LIN {X 0,Y 216.642,Z 888.332,A -85,B 0,C 180,E1 18460.085,E2 18460.085} C_VEL
LIN {X 0,Y 215.367,Z 897.562,A -85,B 0,C 180,E1 18472.801,E2 18472.801} C_VEL
LIN {X 0,Y 221.756,Z 891.791,A -85,B 0,C 180,E1 18485.568,E2 18485.568} C_VEL
LIN {X 0,Y 234.367,Z 872.004,A -85,B 0,C 180,E1 18496.083,E2 18496.083} C_VEL
LIN {X 0,Y 246.425,Z 844.143,A -85,B 0,C 180,E1 18503.35,E2 18503.35} C_VEL
LIN {X 0,Y 242.463,Z 813.223,A -85,B 0,C 180,E1 18511.998,E2 18511.998} C_VEL
LIN {X 0,Y 229.534,Z 783.44,A -85,B 0,C 180,E1 18522.815,E2 18522.815} C_VEL
LIN {X 0,Y 219.501,Z 768.602,A -85,B 0,C 180,E1 18532.547,E2 18532.547} C_VEL
LIN {X 0,Y 216.132,Z 762.311,A -85,B 0,C 180,E1 18538.989,E2 18538.989} C_VEL
LIN {X 0,Y 216.801,Z 764.753,A -85,B 0,C 180,E1 18552.68,E2 18552.68} C_VEL
LIN {X 0,Y 226.089,Z 777.855,A -85,B 0,C 180,E1 18563.686,E2 18563.686} C_VEL
LIN {X 0,Y 243.459,Z 806.862,A -85,B 0,C 180,E1 18574.796,E2 18574.796} C_VEL
LIN {X 0,Y 255.396,Z 841.876,A -85,B 0,C 180,E1 18582.72,E2 18582.72} C_VEL
LIN {X 0,Y 253.54,Z 855.895,A -85,B 0,C 180,E1 18584.51,E2 18584.51} C_VEL
LIN {X 0,Y 237.346,Z 898.415,A -85,B 0,C 180,E1 18590.848,E2 18590.848} C_VEL
LIN {X 0,Y 221.071,Z 933.004,A -85,B 0,C 180,E1 18601.282,E2 18601.282} C_VEL
LIN {X 0,Y 213.369,Z 954.07,A -85,B 0,C 180,E1 18614.546,E2 18614.546} C_VEL
LIN {X 0,Y 214.082,Z 960.88,A -85,B 0,C 180,E1 18627.97,E2 18627.97} C_VEL
LIN {X 0,Y 213.585,Z 955.524,A -85,B 0,C 180,E1 18638.754,E2 18638.754} C_VEL
LIN {X 0,Y 215.65,Z 935.355,A -85,B 0,C 180,E1 18651.683,E2 18651.683} C_VEL
LIN {X 0,Y 225.142,Z 901.268,A -85,B 0,C 180,E1 18662.599,E2 18662.599} C_VEL
LIN {X 0,Y 236.885,Z 857.02,A -85,B 0,C 180,E1 18669.903,E2 18669.903} C_VEL
LIN {X 0,Y 239.376,Z 834.505,A -85,B 0,C 180,E1 18672.297,E2 18672.297} C_VEL
LIN {X 0,Y 223.033,Z 785.451,A -85,B 0,C 180,E1 18678.284,E2 18678.284} C_VEL
LIN {X 0,Y 208.065,Z 754.81,A -85,B 0,C 180,E1 18683.186,E2 18683.186} C_VEL
LIN {X 0,Y 208.631,Z 754.81,A -85,B 0,C 180,E1 18696.424,E2 18696.424} C_VEL
LIN {X 0,Y 209.987,Z 754.81,A -85,B 0,C 180,E1 18709.596,E2 18709.596} C_VEL
LIN {X 0,Y 211.028,Z 754.81,A -85,B 0,C 180,E1 18722.066,E2 18722.066} C_VEL
LIN {X 0,Y 209.557,Z 754.81,A -85,B 0,C 180,E1 18734.688,E2 18734.688} C_VEL
LIN {X 0,Y 208.363,Z 754.81,A -85,B 0,C 180,E1 18748.262,E2 18748.262} C_VEL
LIN {X 0,Y 207.688,Z 754.81,A -85,B 0,C 180,E1 18755.24,E2 18755.24} C_VEL
LIN {X 0,Y 199.559,Z 754.81,A -85,B 0,C 180,E1 18765.026,E2 18765.026} C_VEL
LIN {X 0,Y 200.085,Z 754.81,A -85,B 0,C 180,E1 18780.729,E2 18780.729} C_VEL
LIN {X 0,Y 200.76,Z 756.849,A -85,B 0,C 180,E1 18786.458,E2 18786.458} C_VEL
LIN {X 0,Y 219.95,Z 797.875,A -85,B 0,C 180,E1 18793.889,E2 18793.889} C_VEL
LIN {X 0,Y 225.128,Z 832.107,A -85,B 0,C 180,E1 18800.297,E2 18800.297} C_VEL
LIN {X 0,Y 216.024,Z 866.137,A -85,B 0,C 180,E1 18808.489,E2 18808.489} C_VEL
LIN {X 0,Y 208.947,Z 888.832,A -85,B 0,C 180,E1 18819.404,E2 18819.404} C_VEL
LIN {X 0,Y 207.037,Z 897.624,A -85,B 0,C 180,E1 18829.258,E2 18829.258} C_VEL
LIN {X 0,Y 211.47,Z 896.323,A -85,B 0,C 180,E1 18842.561,E2 18842.561} C_VEL
LIN {X 0,Y 222.672,Z 881.638,A -85,B 0,C 180,E1 18853.742,E2 18853.742} C_VEL
LIN {X 0,Y 238.779,Z 852.504,A -85,B 0,C 180,E1 18862.854,E2 18862.854} C_VEL
LIN {X 0,Y 239.096,Z 827.128,A -85,B 0,C 180,E1 18870.117,E2 18870.117} C_VEL
LIN {X 0,Y 230.039,Z 797.834,A -85,B 0,C 180,E1 18880.234,E2 18880.234} C_VEL
LIN {X 0,Y 218.96,Z 777.151,A -85,B 0,C 180,E1 18891.777,E2 18891.777} C_VEL
LIN {X 0,Y 214.743,Z 770.093,A -85,B 0,C 180,E1 18899.995,E2 18899.995} C_VEL
LIN {X 0,Y 215.607,Z 772.884,A -85,B 0,C 180,E1 18912.422,E2 18912.422} C_VEL
LIN {X 0,Y 224.315,Z 785.804,A -85,B 0,C 180,E1 18923.242,E2 18923.242} C_VEL
LIN {X 0,Y 239.528,Z 813.168,A -85,B 0,C 180,E1 18934.071,E2 18934.071} C_VEL
LIN {X 0,Y 249.646,Z 846.608,A -85,B 0,C 180,E1 18942.026,E2 18942.026} C_VEL
LIN {X 0,Y 234.399,Z 890.534,A -85,B 0,C 180,E1 18948.112,E2 18948.112} C_VEL
LIN {X 0,Y 217.163,Z 925.879,A -85,B 0,C 180,E1 18957.631,E2 18957.631} C_VEL
LIN {X 0,Y 206.591,Z 949.509,A -85,B 0,C 180,E1 18970.699,E2 18970.699} C_VEL
LIN {X 0,Y 205.64,Z 959.398,A -85,B 0,C 180,E1 18984.976,E2 18984.976} C_VEL
LIN {X 0,Y 205.897,Z 956.427,A -85,B 0,C 180,E1 18996.349,E2 18996.349} C_VEL
LIN {X 0,Y 206.874,Z 939.032,A -85,B 0,C 180,E1 19009.834,E2 19009.834} C_VEL
LIN {X 0,Y 215.884,Z 906.703,A -85,B 0,C 180,E1 19021.819,E2 19021.819} C_VEL
LIN {X 0,Y 227.99,Z 864.284,A -85,B 0,C 180,E1 19029.883,E2 19029.883} C_VEL
LIN {X 0,Y 232.17,Z 835.979,A -85,B 0,C 180,E1 19033.141,E2 19033.141} C_VEL
LIN {X 0,Y 216.478,Z 787.844,A -85,B 0,C 180,E1 19039.468,E2 19039.468} C_VEL
LIN {X 0,Y 200.012,Z 754.81,A -85,B 0,C 180,E1 19045.323,E2 19045.323} C_VEL
LIN {X 0,Y 201.013,Z 754.81,A -85,B 0,C 180,E1 19060.687,E2 19060.687} C_VEL
LIN {X 0,Y 202.403,Z 754.81,A -85,B 0,C 180,E1 19073.548,E2 19073.548} C_VEL
LIN {X 0,Y 202.353,Z 754.81,A -85,B 0,C 180,E1 19086.465,E2 19086.465} C_VEL
LIN {X 0,Y 200.993,Z 754.81,A -85,B 0,C 180,E1 19099.868,E2 19099.868} C_VEL
LIN {X 0,Y 199.695,Z 754.81,A -85,B 0,C 180,E1 19115.187,E2 19115.187} C_VEL
LIN {X 0,Y 199.559,Z 754.81,A -85,B 0,C 180,E1 19125.026,E2 19125.026} C_VEL
LIN {X 0,Y 191.609,Z 754.81,A -85,B 0,C 180,E1 19135.197,E2 19135.197} C_VEL
LIN {X 0,Y 192.38,Z 756.459,A -85,B 0,C 180,E1 19144.182,E2 19144.182} C_VEL
LIN {X 0,Y 211.999,Z 796.756,A -85,B 0,C 180,E1 19152.184,E2 19152.184} C_VEL
LIN {X 0,Y 217.973,Z 830.392,A -85,B 0,C 180,E1 19158.773,E2 19158.773} C_VEL
LIN {X 0,Y 209.876,Z 862.822,A -85,B 0,C 180,E1 19166.371,E2 19166.371} C_VEL
LIN {X 0,Y 201.767,Z 887.669,A -85,B 0,C 180,E1 19177.517,E2 19177.517} C_VEL
LIN {X 0,Y 199.152,Z 899.09,A -85,B 0,C 180,E1 19190.053,E2 19190.053} C_VEL
LIN {X 0,Y 204.345,Z 897.187,A -85,B 0,C 180,E1 19203.846,E2 19203.846} C_VEL
LIN {X 0,Y 217.901,Z 879.987,A -85,B 0,C 180,E1 19216.181,E2 19216.181} C_VEL
LIN {X 0,Y 233.671,Z 850.1,A -85,B 0,C 180,E1 19225.187,E2 19225.187} C_VEL
LIN {X 0,Y 231.584,Z 820.81,A -85,B 0,C 180,E1 19234.506,E2 19234.506} C_VEL
LIN {X 0,Y 221.936,Z 794.694,A -85,B 0,C 180,E1 19245.77,E2 19245.77} C_VEL
LIN {X 0,Y 214.394,Z 778.368,A -85,B 0,C 180,E1 19257.967,E2 19257.967} C_VEL
LIN {X 0,Y 214.31,Z 780.597,A -85,B 0,C 180,E1 19271.92,E2 19271.92} C_VEL
LIN {X 0,Y 222.449,Z 793.997,A -85,B 0,C 180,E1 19282.967,E2 19282.967} C_VEL
LIN {X 0,Y 235.748,Z 820.234,A -85,B 0,C 180,E1 19293.604,E2 19293.604} C_VEL
LIN {X 0,Y 243.852,Z 851.713,A -85,B 0,C 180,E1 19301.417,E2 19301.417} C_VEL
LIN {X 0,Y 226.095,Z 894.862,A -85,B 0,C 180,E1 19307.709,E2 19307.709} C_VEL
LIN {X 0,Y 207.49,Z 930.206,A -85,B 0,C 180,E1 19318.594,E2 19318.594} C_VEL
LIN {X 0,Y 198.097,Z 950.734,A -85,B 0,C 180,E1 19332.015,E2 19332.015} C_VEL
LIN {X 0,Y 197.56,Z 957.948,A -85,B 0,C 180,E1 19343.385,E2 19343.385} C_VEL
LIN {X 0,Y 198.021,Z 956.031,A -85,B 0,C 180,E1 19355.118,E2 19355.118} C_VEL
LIN {X 0,Y 198.683,Z 939.873,A -85,B 0,C 180,E1 19369.188,E2 19369.188} C_VEL
LIN {X 0,Y 207.133,Z 909.933,A -85,B 0,C 180,E1 19381.469,E2 19381.469} C_VEL
LIN {X 0,Y 219.913,Z 867.584,A -85,B 0,C 180,E1 19390.314,E2 19390.314} C_VEL
LIN {X 0,Y 225.138,Z 838.311,A -85,B 0,C 180,E1 19393.92,E2 19393.92} C_VEL
LIN {X 0,Y 210.626,Z 791.691,A -85,B 0,C 180,E1 19400.501,E2 19400.501} C_VEL
LIN {X 0,Y 191.887,Z 754.81,A -85,B 0,C 180,E1 19406.991,E2 19406.991} C_VEL
LIN {X 0,Y 192.724,Z 754.81,A -85,B 0,C 180,E1 19419.253,E2 19419.253} C_VEL
LIN {X 0,Y 194.322,Z 754.81,A -85,B 0,C 180,E1 19433.279,E2 19433.279} C_VEL
LIN {X 0,Y 194.279,Z 754.81,A -85,B 0,C 180,E1 19446.734,E2 19446.734} C_VEL
LIN {X 0,Y 192.8,Z 754.81,A -85,B 0,C 180,E1 19460.75,E2 19460.75} C_VEL
LIN {X 0,Y 191.639,Z 754.81,A -85,B 0,C 180,E1 19476.442,E2 19476.442} C_VEL
LIN {X 0,Y 191.645,Z 754.81,A -85,B 0,C 180,E1 19493.564,E2 19493.564} C_VEL
LIN {X 0,Y 191.609,Z 754.81,A -85,B 0,C 180,E1 19495.197,E2 19495.197} C_VEL
LIN {X 0,Y 183.731,Z 754.81,A -85,B 0,C 180,E1 19499.208,E2 19499.208} C_VEL
LIN {X 0,Y 184.236,Z 756.635,A -85,B 0,C 180,E1 19501.717,E2 19501.717} C_VEL
LIN {X 0,Y 203.8,Z 794.802,A -85,B 0,C 180,E1 19510.168,E2 19510.168} C_VEL
LIN {X 0,Y 210.927,Z 830.344,A -85,B 0,C 180,E1 19517.504,E2 19517.504} C_VEL
LIN {X 0,Y 204.215,Z 859.007,A -85,B 0,C 180,E1 19524.134,E2 19524.134} C_VEL
LIN {X 0,Y 194.675,Z 886.406,A -85,B 0,C 180,E1 19535.591,E2 19535.591} C_VEL
LIN {X 0,Y 191.171,Z 899.454,A -85,B 0,C 180,E1 19548.437,E2 19548.437} C_VEL
LIN {X 0,Y 195.686,Z 899.486,A -85,B 0,C 180,E1 19562.877,E2 19562.877} C_VEL
LIN {X 0,Y 208.51,Z 885.123,A -85,B 0,C 180,E1 19575.477,E2 19575.477} C_VEL
LIN {X 0,Y 225.786,Z 857.601,A -85,B 0,C 180,E1 19584.905,E2 19584.905} C_VEL
LIN {X 0,Y 227.56,Z 833.221,A -85,B 0,C 180,E1 19592.776,E2 19592.776} C_VEL
LIN {X 0,Y 221.295,Z 807.811,A -85,B 0,C 180,E1 19603.05,E2 19603.05} C_VEL
LIN {X 0,Y 213.936,Z 790.965,A -85,B 0,C 180,E1 19614.525,E2 19614.525} C_VEL
LIN {X 0,Y 212.043,Z 785.811,A -85,B 0,C 180,E1 19621.02,E2 19621.02} C_VEL
LIN {X 0,Y 212.903,Z 788.641,A -85,B 0,C 180,E1 19631.751,E2 19631.751} C_VEL
LIN {X 0,Y 220.234,Z 801.886,A -85,B 0,C 180,E1 19642.689,E2 19642.689} C_VEL
LIN {X 0,Y 231.995,Z 827.726,A -85,B 0,C 180,E1 19653.366,E2 19653.366} C_VEL
LIN {X 0,Y 237.051,Z 855.918,A -85,B 0,C 180,E1 19660.426,E2 19660.426} C_VEL
LIN {X 0,Y 217.838,Z 898.908,A -85,B 0,C 180,E1 19667.307,E2 19667.307} C_VEL
LIN {X 0,Y 199.27,Z 931.565,A -85,B 0,C 180,E1 19678.429,E2 19678.429} C_VEL
LIN {X 0,Y 189.619,Z 951.846,A -85,B 0,C 180,E1 19693.734,E2 19693.734} C_VEL
LIN {X 0,Y 190.23,Z 957.232,A -85,B 0,C 180,E1 19707.715,E2 19707.715} C_VEL
LIN {X 0,Y 189.591,Z 950.728,A -85,B 0,C 180,E1 19720.377,E2 19720.377} C_VEL
LIN {X 0,Y 193.25,Z 928.656,A -85,B 0,C 180,E1 19734.969,E2 19734.969} C_VEL
LIN {X 0,Y 204.698,Z 893.624,A -85,B 0,C 180,E1 19746.379,E2 19746.379} C_VEL
LIN {X 0,Y 217.917,Z 847.797,A -85,B 0,C 180,E1 19753.779,E2 19753.779} C_VEL
LIN {X 0,Y 209.733,Z 808.336,A -85,B 0,C 180,E1 19759.633,E2 19759.633} C_VEL
LIN {X 0,Y 186.372,Z 760.571,A -85,B 0,C 180,E1 19768.233,E2 19768.233} C_VEL
LIN {X 0,Y 183.924,Z 754.81,A -85,B 0,C 180,E1 19770.042,E2 19770.042} C_VEL
LIN {X 0,Y 185.05,Z 754.81,A -85,B 0,C 180,E1 19783.326,E2 19783.326} C_VEL
LIN {X 0,Y 186.802,Z 754.81,A -85,B 0,C 180,E1 19797.678,E2 19797.678} C_VEL
LIN {X 0,Y 185.727,Z 754.81,A -85,B 0,C 180,E1 19811.793,E2 19811.793} C_VEL
LIN {X 0,Y 184.071,Z 754.81,A -85,B 0,C 180,E1 19826.971,E2 19826.971} C_VEL
LIN {X 0,Y 183.347,Z 754.81,A -85,B 0,C 180,E1 19844.72,E2 19844.72} C_VEL
LIN {X 0,Y 183.731,Z 754.81,A -85,B 0,C 180,E1 19859.208,E2 19859.208} C_VEL
LIN {X 0,Y 186.245,Z 763.492,A -85,B 0,C 180,E1 19862.685,E2 19862.685} C_VEL
LIN {X 0,Y 191.204,Z 782.709,A -85,B 0,C 180,E1 19865.652,E2 19865.652} C_VEL
LIN {X 0,Y 202.789,Z 819.29,A -85,B 0,C 180,E1 19873.694,E2 19873.694} C_VEL
LIN {X 0,Y 201.736,Z 846.339,A -85,B 0,C 180,E1 19879.748,E2 19879.748} C_VEL
LIN {X 0,Y 190.445,Z 878.405,A -85,B 0,C 180,E1 19890.153,E2 19890.153} C_VEL
LIN {X 0,Y 183.865,Z 896.903,A -85,B 0,C 180,E1 19903.118,E2 19903.118} C_VEL
LIN {X 0,Y 184.797,Z 902.481,A -85,B 0,C 180,E1 19916.849,E2 19916.849} C_VEL
LIN {X 0,Y 195.151,Z 894.31,A -85,B 0,C 180,E1 19931.374,E2 19931.374} C_VEL
LIN {X 0,Y 212.21,Z 872.098,A -85,B 0,C 180,E1 19942.65,E2 19942.65} C_VEL
LIN {X 0,Y 221.528,Z 853.18,A -85,B 0,C 180,E1 19948.193,E2 19948.193} C_VEL
LIN {X 0,Y 220.459,Z 825.911,A -85,B 0,C 180,E1 19958.323,E2 19958.323} C_VEL
LIN {X 0,Y 213.555,Z 802.898,A -85,B 0,C 180,E1 19970.794,E2 19970.794} C_VEL
LIN {X 0,Y 210.375,Z 793.636,A -85,B 0,C 180,E1 19980.929,E2 19980.929} C_VEL
LIN {X 0,Y 211.106,Z 796.544,A -85,B 0,C 180,E1 19991.517,E2 19991.517} C_VEL
LIN {X 0,Y 217.693,Z 809.685,A -85,B 0,C 180,E1 20002.449,E2 20002.449} C_VEL
LIN {X 0,Y 227.555,Z 834.107,A -85,B 0,C 180,E1 20012.806,E2 20012.806} C_VEL
LIN {X 0,Y 231.22,Z 857.687,A -85,B 0,C 180,E1 20019.123,E2 20019.123} C_VEL
LIN {X 0,Y 211.548,Z 899.02,A -85,B 0,C 180,E1 20025.984,E2 20025.984} C_VEL
LIN {X 0,Y 191.672,Z 931.777,A -85,B 0,C 180,E1 20037.696,E2 20037.696} C_VEL
LIN {X 0,Y 181.601,Z 951.475,A -85,B 0,C 180,E1 20053.923,E2 20053.923} C_VEL
LIN {X 0,Y 182.292,Z 956.015,A -85,B 0,C 180,E1 20067.616,E2 20067.616} C_VEL
LIN {X 0,Y 181.721,Z 950.328,A -85,B 0,C 180,E1 20079.616,E2 20079.616} C_VEL
LIN {X 0,Y 184.679,Z 930.394,A -85,B 0,C 180,E1 20094.23,E2 20094.23} C_VEL
LIN {X 0,Y 196.232,Z 896.463,A -85,B 0,C 180,E1 20106.48,E2 20106.48} C_VEL
LIN {X 0,Y 209.934,Z 852.254,A -85,B 0,C 180,E1 20114.357,E2 20114.357} C_VEL
LIN {X 0,Y 209.002,Z 831.793,A -85,B 0,C 180,E1 20117.414,E2 20117.414} C_VEL
LIN {X 0,Y 193.105,Z 786.695,A -85,B 0,C 180,E1 20124.963,E2 20124.963} C_VEL
LIN {X 0,Y 176.04,Z 754.81,A -85,B 0,C 180,E1 20132.545,E2 20132.545} C_VEL
LIN {X 0,Y 177.688,Z 754.81,A -85,B 0,C 180,E1 20149.175,E2 20149.175} C_VEL
LIN {X 0,Y 178.858,Z 754.81,A -85,B 0,C 180,E1 20162.438,E2 20162.438} C_VEL
LIN {X 0,Y 177.009,Z 754.81,A -85,B 0,C 180,E1 20177.468,E2 20177.468} C_VEL
LIN {X 0,Y 175.399,Z 754.81,A -85,B 0,C 180,E1 20194.717,E2 20194.717} C_VEL
LIN {X 0,Y 175.178,Z 754.81,A -85,B 0,C 180,E1 20209.477,E2 20209.477} C_VEL
LIN {X 0,Y 175.877,Z 756.396,A -85,B 0,C 180,E1 20218.796,E2 20218.796} C_VEL
LIN {X 0,Y 191.204,Z 782.709,A -85,B 0,C 180,E1 20225.652,E2 20225.652} C_VEL
LIN {X 0,Y 194.539,Z 813.73,A -85,B 0,C 180,E1 20230.805,E2 20230.805} C_VEL
LIN {X 0,Y 196.081,Z 842.903,A -85,B 0,C 180,E1 20237.716,E2 20237.716} C_VEL
LIN {X 0,Y 184.277,Z 875.529,A -85,B 0,C 180,E1 20247.639,E2 20247.639} C_VEL
LIN {X 0,Y 176.592,Z 896.01,A -85,B 0,C 180,E1 20260.798,E2 20260.798} C_VEL
LIN {X 0,Y 176.358,Z 903.64,A -85,B 0,C 180,E1 20275.361,E2 20275.361} C_VEL
LIN {X 0,Y 186.16,Z 897.498,A -85,B 0,C 180,E1 20290.699,E2 20290.699} C_VEL
LIN {X 0,Y 204.093,Z 876.474,A -85,B 0,C 180,E1 20303.025,E2 20303.025} C_VEL
LIN {X 0,Y 215.35,Z 856.378,A -85,B 0,C 180,E1 20309.262,E2 20309.262} C_VEL
LIN {X 0,Y 215.666,Z 832.062,A -85,B 0,C 180,E1 20318.855,E2 20318.855} C_VEL
LIN {X 0,Y 210.513,Z 809.89,A -85,B 0,C 180,E1 20331.432,E2 20331.432} C_VEL
LIN {X 0,Y 208.183,Z 801.185,A -85,B 0,C 180,E1 20342.083,E2 20342.083} C_VEL
LIN {X 0,Y 208.98,Z 804.42,A -85,B 0,C 180,E1 20351.385,E2 20351.385} C_VEL
LIN {X 0,Y 214.51,Z 816.583,A -85,B 0,C 180,E1 20361.797,E2 20361.797} C_VEL
LIN {X 0,Y 222.765,Z 839.779,A -85,B 0,C 180,E1 20372.04,E2 20372.04} C_VEL
LIN {X 0,Y 224.498,Z 861.643,A -85,B 0,C 180,E1 20378.011,E2 20378.011} C_VEL
LIN {X 0,Y 203.15,Z 902.913,A -85,B 0,C 180,E1 20385.548,E2 20385.548} C_VEL
LIN {X 0,Y 183.452,Z 932.959,A -85,B 0,C 180,E1 20397.474,E2 20397.474} C_VEL
LIN {X 0,Y 173.684,Z 950.664,A -85,B 0,C 180,E1 20413.637,E2 20413.637} C_VEL
LIN {X 0,Y 174.339,Z 954.776,A -85,B 0,C 180,E1 20427.507,E2 20427.507} C_VEL
LIN {X 0,Y 173.756,Z 948.862,A -85,B 0,C 180,E1 20440.062,E2 20440.062} C_VEL
LIN {X 0,Y 177.417,Z 927.956,A -85,B 0,C 180,E1 20455.624,E2 20455.624} C_VEL
LIN {X 0,Y 189.677,Z 893.977,A -85,B 0,C 180,E1 20467.959,E2 20467.959} C_VEL
LIN {X 0,Y 203.64,Z 850.097,A -85,B 0,C 180,E1 20475.748,E2 20475.748} C_VEL
LIN {X 0,Y 196.001,Z 811.221,A -85,B 0,C 180,E1 20482.437,E2 20482.437} C_VEL
LIN {X 0,Y 174.661,Z 766.987,A -85,B 0,C 180,E1 20491.859,E2 20491.859} C_VEL
LIN {X 0,Y 168.178,Z 754.81,A -85,B 0,C 180,E1 20496.05,E2 20496.05} C_VEL
LIN {X 0,Y 170.064,Z 754.81,A -85,B 0,C 180,E1 20512.314,E2 20512.314} C_VEL
LIN {X 0,Y 170.796,Z 754.81,A -85,B 0,C 180,E1 20522.553,E2 20522.553} C_VEL
LIN {X 0,Y 168.649,Z 754.81,A -85,B 0,C 180,E1 20539.115,E2 20539.115} C_VEL
LIN {X 0,Y 167.173,Z 754.81,A -85,B 0,C 180,E1 20556.169,E2 20556.169} C_VEL
LIN {X 0,Y 167.158,Z 754.81,A -85,B 0,C 180,E1 20573.833,E2 20573.833} C_VEL
LIN {X 0,Y 168.298,Z 758.387,A -85,B 0,C 180,E1 20575.922,E2 20575.922} C_VEL
LIN {X 0,Y 187.651,Z 792.072,A -85,B 0,C 180,E1 20585.695,E2 20585.695} C_VEL
LIN {X 0,Y 194.539,Z 813.73,A -85,B 0,C 180,E1 20590.805,E2 20590.805} C_VEL
LIN {X 0,Y 191.602,Z 836.321,A -85,B 0,C 180,E1 20595.002,E2 20595.002} C_VEL
LIN {X 0,Y 189.261,Z 843.612,A -85,B 0,C 180,E1 20596.494,E2 20596.494} C_VEL
LIN {X 0,Y 176.72,Z 876.776,A -85,B 0,C 180,E1 20606.922,E2 20606.922} C_VEL
LIN {X 0,Y 168.388,Z 898.052,A -85,B 0,C 180,E1 20621.546,E2 20621.546} C_VEL
LIN {X 0,Y 168.057,Z 904.57,A -85,B 0,C 180,E1 20633.974,E2 20633.974} C_VEL
LIN {X 0,Y 177.177,Z 900.405,A -85,B 0,C 180,E1 20649.969,E2 20649.969} C_VEL
LIN {X 0,Y 195.65,Z 881.029,A -85,B 0,C 180,E1 20663.258,E2 20663.258} C_VEL
LIN {X 0,Y 209.024,Z 860.383,A -85,B 0,C 180,E1 20670.037,E2 20670.037} C_VEL
LIN {X 0,Y 210.464,Z 835.648,A -85,B 0,C 180,E1 20680.514,E2 20680.514} C_VEL
LIN {X 0,Y 206.875,Z 814.753,A -85,B 0,C 180,E1 20693.677,E2 20693.677} C_VEL
LIN {X 0,Y 205.811,Z 808.827,A -85,B 0,C 180,E1 20702.107,E2 20702.107} C_VEL
LIN {X 0,Y 206.426,Z 811.438,A -85,B 0,C 180,E1 20710.585,E2 20710.585} C_VEL
LIN {X 0,Y 212.449,Z 826.515,A -85,B 0,C 180,E1 20723.128,E2 20723.128} C_VEL
LIN {X 0,Y 218.908,Z 852.529,A -85,B 0,C 180,E1 20733.676,E2 20733.676} C_VEL
LIN {X 0,Y 217.99,Z 865.134,A -85,B 0,C 180,E1 20736.816,E2 20736.816} C_VEL
LIN {X 0,Y 195.266,Z 905.655,A -85,B 0,C 180,E1 20744.834,E2 20744.834} C_VEL
LIN {X 0,Y 175.235,Z 933.977,A -85,B 0,C 180,E1 20757.232,E2 20757.232} C_VEL
LIN {X 0,Y 165.619,Z 950.321,A -85,B 0,C 180,E1 20774.151,E2 20774.151} C_VEL
LIN {X 0,Y 166.391,Z 953.516,A -85,B 0,C 180,E1 20787.388,E2 20787.388} C_VEL
LIN {X 0,Y 165.799,Z 947.396,A -85,B 0,C 180,E1 20800.55,E2 20800.55} C_VEL
LIN {X 0,Y 170.473,Z 925.115,A -85,B 0,C 180,E1 20817.316,E2 20817.316} C_VEL
LIN {X 0,Y 184.074,Z 889.049,A -85,B 0,C 180,E1 20830.099,E2 20830.099} C_VEL
LIN {X 0,Y 196.926,Z 846.331,A -85,B 0,C 180,E1 20837.595,E2 20837.595} C_VEL
LIN {X 0,Y 185.511,Z 802.686,A -85,B 0,C 180,E1 20845.962,E2 20845.962} C_VEL
LIN {X 0,Y 163.671,Z 761.429,A -85,B 0,C 180,E1 20856.8,E2 20856.8} C_VEL
LIN {X 0,Y 160.397,Z 754.81,A -85,B 0,C 180,E1 20859.922,E2 20859.922} C_VEL
LIN {X 0,Y 162.642,Z 754.81,A -85,B 0,C 180,E1 20877.333,E2 20877.333} C_VEL
LIN {X 0,Y 161.263,Z 754.81,A -85,B 0,C 180,E1 20893.614,E2 20893.614} C_VEL
LIN {X 0,Y 159.331,Z 754.81,A -85,B 0,C 180,E1 20911.599,E2 20911.599} C_VEL
LIN {X 0,Y 159.086,Z 754.81,A -85,B 0,C 180,E1 20930.981,E2 20930.981} C_VEL
LIN {X 0,Y 180.674,Z 792.986,A -85,B 0,C 180,E1 20943.716,E2 20943.716} C_VEL
LIN {X 0,Y 189.657,Z 828.357,A -85,B 0,C 180,E1 20952.637,E2 20952.637} C_VEL
LIN {X 0,Y 189.261,Z 843.612,A -85,B 0,C 180,E1 20956.494,E2 20956.494} C_VEL
LIN {X 0,Y 176.1,Z 861.099,A -85,B 0,C 180,E1 20959.584,E2 20959.584} C_VEL
LIN {X 0,Y 164.15,Z 889.393,A -85,B 0,C 180,E1 20972.648,E2 20972.648} C_VEL
LIN {X 0,Y 159.509,Z 904.247,A -85,B 0,C 180,E1 20989.449,E2 20989.449} C_VEL
LIN {X 0,Y 165.978,Z 904.412,A -85,B 0,C 180,E1 21006.461,E2 21006.461} C_VEL
LIN {X 0,Y 182.01,Z 890.921,A -85,B 0,C 180,E1 21020.464,E2 21020.464} C_VEL
LIN {X 0,Y 202.726,Z 864.295,A -85,B 0,C 180,E1 21030.878,E2 21030.878} C_VEL
LIN {X 0,Y 205.475,Z 841.52,A -85,B 0,C 180,E1 21041.143,E2 21041.143} C_VEL
LIN {X 0,Y 203.581,Z 822.517,A -85,B 0,C 180,E1 21053.575,E2 21053.575} C_VEL
LIN {X 0,Y 203.096,Z 816.34,A -85,B 0,C 180,E1 21062.136,E2 21062.136} C_VEL
LIN {X 0,Y 203.666,Z 819.259,A -85,B 0,C 180,E1 21070.73,E2 21070.73} C_VEL
LIN {X 0,Y 209.091,Z 835.017,A -85,B 0,C 180,E1 21083.521,E2 21083.521} C_VEL
LIN {X 0,Y 213.695,Z 860.972,A -85,B 0,C 180,E1 21094.021,E2 21094.021} C_VEL
LIN {X 0,Y 205.868,Z 879.022,A -85,B 0,C 180,E1 21097.153,E2 21097.153} C_VEL
LIN {X 0,Y 182.218,Z 915.381,A -85,B 0,C 180,E1 21106.602,E2 21106.602} C_VEL
LIN {X 0,Y 163.126,Z 940.117,A -85,B 0,C 180,E1 21121.322,E2 21121.322} C_VEL
LIN {X 0,Y 157.45,Z 950.424,A -85,B 0,C 180,E1 21136.059,E2 21136.059} C_VEL
LIN {X 0,Y 158.42,Z 952.251,A -85,B 0,C 180,E1 21147.256,E2 21147.256} C_VEL
LIN {X 0,Y 157.833,Z 945.921,A -85,B 0,C 180,E1 21161.089,E2 21161.089} C_VEL
LIN {X 0,Y 162.527,Z 924.936,A -85,B 0,C 180,E1 21177.688,E2 21177.688} C_VEL
LIN {X 0,Y 176.518,Z 889.69,A -85,B 0,C 180,E1 21190.963,E2 21190.963} C_VEL
LIN {X 0,Y 189.895,Z 847.707,A -85,B 0,C 180,E1 21198.756,E2 21198.756} C_VEL
LIN {X 0,Y 179.095,Z 804.623,A -85,B 0,C 180,E1 21207.671,E2 21207.671} C_VEL
LIN {X 0,Y 159.297,Z 767.1,A -85,B 0,C 180,E1 21218.527,E2 21218.527} C_VEL
LIN {X 0,Y 152.647,Z 754.81,A -85,B 0,C 180,E1 21223.46,E2 21223.46} C_VEL
LIN {X 0,Y 154.577,Z 754.81,A -85,B 0,C 180,E1 21237.194,E2 21237.194} C_VEL
LIN {X 0,Y 153.839,Z 754.81,A -85,B 0,C 180,E1 21248.516,E2 21248.516} C_VEL
LIN {X 0,Y 151.619,Z 754.81,A -85,B 0,C 180,E1 21266.778,E2 21266.778} C_VEL
LIN {X 0,Y 151.268,Z 756.664,A -85,B 0,C 180,E1 21286.83,E2 21286.83} C_VEL
LIN {X 0,Y 171.817,Z 789.685,A -85,B 0,C 180,E1 21300.214,E2 21300.214} C_VEL
LIN {X 0,Y 182.257,Z 824.923,A -85,B 0,C 180,E1 21309.981,E2 21309.981} C_VEL
LIN {X 0,Y 180.809,Z 849.295,A -85,B 0,C 180,E1 21316.344,E2 21316.344} C_VEL
LIN {X 0,Y 176.1,Z 861.099,A -85,B 0,C 180,E1 21319.584,E2 21319.584} C_VEL
LIN {X 0,Y 159.921,Z 883.072,A -85,B 0,C 180,E1 21327.32,E2 21327.32} C_VEL
LIN {X 0,Y 152.131,Z 901.642,A -85,B 0,C 180,E1 21342.969,E2 21342.969} C_VEL
LIN {X 0,Y 152.869,Z 907.155,A -85,B 0,C 180,E1 21356.532,E2 21356.532} C_VEL
LIN {X 0,Y 164.565,Z 901.89,A -85,B 0,C 180,E1 21373.757,E2 21373.757} C_VEL
LIN {X 0,Y 185.284,Z 882.217,A -85,B 0,C 180,E1 21387.088,E2 21387.088} C_VEL
LIN {X 0,Y 197.194,Z 865.618,A -85,B 0,C 180,E1 21392.914,E2 21392.914} C_VEL
LIN {X 0,Y 200.431,Z 844.135,A -85,B 0,C 180,E1 21403.498,E2 21403.498} C_VEL
LIN {X 0,Y 199.742,Z 828.068,A -85,B 0,C 180,E1 21415.637,E2 21415.637} C_VEL
LIN {X 0,Y 200.035,Z 823.739,A -85,B 0,C 180,E1 21422.168,E2 21422.168} C_VEL
LIN {X 0,Y 201.072,Z 828.649,A -85,B 0,C 180,E1 21433.081,E2 21433.081} C_VEL
LIN {X 0,Y 205.924,Z 846.391,A -85,B 0,C 180,E1 21445.51,E2 21445.51} C_VEL
LIN {X 0,Y 207.413,Z 867.462,A -85,B 0,C 180,E1 21453.619,E2 21453.619} C_VEL
LIN {X 0,Y 182.477,Z 906.789,A -85,B 0,C 180,E1 21461.949,E2 21461.949} C_VEL
LIN {X 0,Y 160.222,Z 933.989,A -85,B 0,C 180,E1 21475.37,E2 21475.37} C_VEL
LIN {X 0,Y 149.56,Z 949.304,A -85,B 0,C 180,E1 21495.307,E2 21495.307} C_VEL
LIN {X 0,Y 150.457,Z 950.983,A -85,B 0,C 180,E1 21507.111,E2 21507.111} C_VEL
LIN {X 0,Y 149.89,Z 944.409,A -85,B 0,C 180,E1 21521.685,E2 21521.685} C_VEL
LIN {X 0,Y 155.567,Z 922.122,A -85,B 0,C 180,E1 21539.553,E2 21539.553} C_VEL
LIN {X 0,Y 170.855,Z 885.883,A -85,B 0,C 180,E1 21553.067,E2 21553.067} C_VEL
LIN {X 0,Y 182.756,Z 847.533,A -85,B 0,C 180,E1 21560.339,E2 21560.339} C_VEL
LIN {X 0,Y 172.166,Z 804.963,A -85,B 0,C 180,E1 21569.92,E2 21569.92} C_VEL
LIN {X 0,Y 152.674,Z 767.998,A -85,B 0,C 180,E1 21582.122,E2 21582.122} C_VEL
LIN {X 0,Y 145.369,Z 754.81,A -85,B 0,C 180,E1 21589.481,E2 21589.481} C_VEL
LIN {X 0,Y 146.6,Z 754.81,A -85,B 0,C 180,E1 21602.974,E2 21602.974} C_VEL
LIN {X 0,Y 144.028,Z 754.81,A -85,B 0,C 180,E1 21621.648,E2 21621.648} C_VEL
LIN {X 0,Y 143.05,Z 756.69,A -85,B 0,C 180,E1 21640.534,E2 21640.534} C_VEL
LIN {X 0,Y 160.523,Z 782.457,A -85,B 0,C 180,E1 21654.545,E2 21654.545} C_VEL
LIN {X 0,Y 173.178,Z 814.038,A -85,B 0,C 180,E1 21664.906,E2 21664.906} C_VEL
LIN {X 0,Y 175.69,Z 844.811,A -85,B 0,C 180,E1 21673.665,E2 21673.665} C_VEL
LIN {X 0,Y 161.656,Z 879.225,A -85,B 0,C 180,E1 21685.287,E2 21685.287} C_VEL
LIN {X 0,Y 159.921,Z 883.072,A -85,B 0,C 180,E1 21687.32,E2 21687.32} C_VEL
LIN {X 0,Y 145.616,Z 898.896,A -85,B 0,C 180,E1 21697.984,E2 21697.984} C_VEL
LIN {X 0,Y 145.137,Z 908.357,A -85,B 0,C 180,E1 21717.266,E2 21717.266} C_VEL
LIN {X 0,Y 158.544,Z 902.637,A -85,B 0,C 180,E1 21735.879,E2 21735.879} C_VEL
LIN {X 0,Y 180.654,Z 882.601,A -85,B 0,C 180,E1 21749.248,E2 21749.248} C_VEL
LIN {X 0,Y 191.59,Z 867.693,A -85,B 0,C 180,E1 21754.728,E2 21754.728} C_VEL
LIN {X 0,Y 195.463,Z 847.846,A -85,B 0,C 180,E1 21765.493,E2 21765.493} C_VEL
LIN {X 0,Y 196.073,Z 833.601,A -85,B 0,C 180,E1 21777.901,E2 21777.901} C_VEL
LIN {X 0,Y 196.923,Z 831.364,A -85,B 0,C 180,E1 21786.632,E2 21786.632} C_VEL
LIN {X 0,Y 199.508,Z 844.093,A -85,B 0,C 180,E1 21800.011,E2 21800.011} C_VEL
LIN {X 0,Y 202.131,Z 866.241,A -85,B 0,C 180,E1 21810.886,E2 21810.886} C_VEL
LIN {X 0,Y 197.349,Z 877.201,A -85,B 0,C 180,E1 21813.202,E2 21813.202} C_VEL
LIN {X 0,Y 170.706,Z 914.09,A -85,B 0,C 180,E1 21822.828,E2 21822.828} C_VEL
LIN {X 0,Y 148.147,Z 939.059,A -85,B 0,C 180,E1 21839.196,E2 21839.196} C_VEL
LIN {X 0,Y 141.603,Z 949.592,A -85,B 0,C 180,E1 21860.751,E2 21860.751} C_VEL
LIN {X 0,Y 142.716,Z 948.254,A -85,B 0,C 180,E1 21873.05,E2 21873.05} C_VEL
LIN {X 0,Y 143.42,Z 933.81,A -85,B 0,C 180,E1 21891.739,E2 21891.739} C_VEL
LIN {X 0,Y 155.658,Z 904.308,A -85,B 0,C 180,E1 21908.43,E2 21908.43} C_VEL
LIN {X 0,Y 172.494,Z 863.722,A -85,B 0,C 180,E1 21919.053,E2 21919.053} C_VEL
LIN {X 0,Y 175.696,Z 847.804,A -85,B 0,C 180,E1 21921.946,E2 21921.946} C_VEL
LIN {X 0,Y 166.062,Z 807.238,A -85,B 0,C 180,E1 21931.86,E2 21931.86} C_VEL
LIN {X 0,Y 148.603,Z 773.389,A -85,B 0,C 180,E1 21944.216,E2 21944.216} C_VEL
LIN {X 0,Y 138.422,Z 754.81,A -85,B 0,C 180,E1 21956.866,E2 21956.866} C_VEL
LIN {X 0,Y 137.518,Z 754.81,A -85,B 0,C 180,E1 21969.536,E2 21969.536} C_VEL
LIN {X 0,Y 135.005,Z 754.81,A -85,B 0,C 180,E1 21990.396,E2 21990.396} C_VEL
LIN {X 0,Y 149.457,Z 776.548,A -85,B 0,C 180,E1 22007.689,E2 22007.689} C_VEL
LIN {X 0,Y 163.81,Z 805.779,A -85,B 0,C 180,E1 22019.834,E2 22019.834} C_VEL
LIN {X 0,Y 169.528,Z 838.575,A -85,B 0,C 180,E1 22030.057,E2 22030.057} C_VEL
LIN {X 0,Y 163.522,Z 859.776,A -85,B 0,C 180,E1 22036.033,E2 22036.033} C_VEL
LIN {X 0,Y 149.567,Z 889.758,A -85,B 0,C 180,E1 22049.998,E2 22049.998} C_VEL
LIN {X 0,Y 145.616,Z 898.896,A -85,B 0,C 180,E1 22057.984,E2 22057.984} C_VEL
LIN {X 0,Y 135.891,Z 908.043,A -85,B 0,C 180,E1 22071.414,E2 22071.414} C_VEL
LIN {X 0,Y 143.649,Z 908.396,A -85,B 0,C 180,E1 22089.33,E2 22089.33} C_VEL
LIN {X 0,Y 163.43,Z 895.288,A -85,B 0,C 180,E1 22105.292,E2 22105.292} C_VEL
LIN {X 0,Y 185.246,Z 872.028,A -85,B 0,C 180,E1 22115.504,E2 22115.504} C_VEL
LIN {X 0,Y 190.37,Z 853.337,A -85,B 0,C 180,E1 22126.327,E2 22126.327} C_VEL
LIN {X 0,Y 192.089,Z 840.653,A -85,B 0,C 180,E1 22137.964,E2 22137.964} C_VEL
LIN {X 0,Y 193.211,Z 838.625,A -85,B 0,C 180,E1 22146.76,E2 22146.76} C_VEL
LIN {X 0,Y 195.317,Z 851.814,A -85,B 0,C 180,E1 22160.459,E2 22160.459} C_VEL
LIN {X 0,Y 196.288,Z 871.204,A -85,B 0,C 180,E1 22170.161,E2 22170.161} C_VEL
LIN {X 0,Y 168.781,Z 909.485,A -85,B 0,C 180,E1 22179.23,E2 22179.23} C_VEL
LIN {X 0,Y 143.906,Z 935.37,A -85,B 0,C 180,E1 22194.551,E2 22194.551} C_VEL
LIN {X 0,Y 133.746,Z 947.32,A -85,B 0,C 180,E1 22214.645,E2 22214.645} C_VEL
LIN {X 0,Y 134.504,Z 948.441,A -85,B 0,C 180,E1 22226.768,E2 22226.768} C_VEL
LIN {X 0,Y 134.033,Z 942.542,A -85,B 0,C 180,E1 22241.387,E2 22241.387} C_VEL
LIN {X 0,Y 140.602,Z 919.962,A -85,B 0,C 180,E1 22261.75,E2 22261.75} C_VEL
LIN {X 0,Y 157.135,Z 884.816,A -85,B 0,C 180,E1 22275.917,E2 22275.917} C_VEL
LIN {X 0,Y 169.104,Z 851.827,A -85,B 0,C 180,E1 22282.726,E2 22282.726} C_VEL
LIN {X 0,Y 160.892,Z 811.959,A -85,B 0,C 180,E1 22293.21,E2 22293.21} C_VEL
LIN {X 0,Y 145.411,Z 779.496,A -85,B 0,C 180,E1 22305.85,E2 22305.85} C_VEL
LIN {X 0,Y 134.592,Z 761.91,A -85,B 0,C 180,E1 22319.201,E2 22319.201} C_VEL
LIN {X 0,Y 129.869,Z 759.669,A -85,B 0,C 180,E1 22338.312,E2 22338.312} C_VEL
LIN {X 0,Y 133.773,Z 765.444,A -85,B 0,C 180,E1 22351.135,E2 22351.135} C_VEL
LIN {X 0,Y 143.768,Z 779.399,A -85,B 0,C 180,E1 22364.043,E2 22364.043} C_VEL
LIN {X 0,Y 157.043,Z 806.476,A -85,B 0,C 180,E1 22377.085,E2 22377.085} C_VEL
LIN {X 0,Y 162.793,Z 837.73,A -85,B 0,C 180,E1 22387.709,E2 22387.709} C_VEL
LIN {X 0,Y 158.424,Z 857.016,A -85,B 0,C 180,E1 22393.435,E2 22393.435} C_VEL
LIN {X 0,Y 143.628,Z 887.696,A -85,B 0,C 180,E1 22406.97,E2 22406.97} C_VEL
LIN {X 0,Y 136.245,Z 903.988,A -85,B 0,C 180,E1 22422.87,E2 22422.87} C_VEL
LIN {X 0,Y 135.891,Z 908.043,A -85,B 0,C 180,E1 22431.414,E2 22431.414} C_VEL
LIN {X 0,Y 133.42,Z 910.457,A -85,B 0,C 180,E1 22446.497,E2 22446.497} C_VEL
LIN {X 0,Y 151.32,Z 901.376,A -85,B 0,C 180,E1 22463.441,E2 22463.441} C_VEL
LIN {X 0,Y 177.552,Z 877.749,A -85,B 0,C 180,E1 22475.845,E2 22475.845} C_VEL
LIN {X 0,Y 184.457,Z 861.758,A -85,B 0,C 180,E1 22484.985,E2 22484.985} C_VEL
LIN {X 0,Y 187.782,Z 847.52,A -85,B 0,C 180,E1 22498.055,E2 22498.055} C_VEL
LIN {X 0,Y 189.166,Z 845.719,A -85,B 0,C 180,E1 22506.906,E2 22506.906} C_VEL
LIN {X 0,Y 190.469,Z 857.766,A -85,B 0,C 180,E1 22519.786,E2 22519.786} C_VEL
LIN {X 0,Y 189.678,Z 875.703,A -85,B 0,C 180,E1 22528.954,E2 22528.954} C_VEL
LIN {X 0,Y 161.322,Z 911.552,A -85,B 0,C 180,E1 22538.018,E2 22538.018} C_VEL
LIN {X 0,Y 135.763,Z 935.864,A -85,B 0,C 180,E1 22554.069,E2 22554.069} C_VEL
LIN {X 0,Y 126.056,Z 945.87,A -85,B 0,C 180,E1 22572.486,E2 22572.486} C_VEL
LIN {X 0,Y 126.523,Z 947.165,A -85,B 0,C 180,E1 22586.564,E2 22586.564} C_VEL
LIN {X 0,Y 126.096,Z 941.133,A -85,B 0,C 180,E1 22601.953,E2 22601.953} C_VEL
LIN {X 0,Y 133.063,Z 919.207,A -85,B 0,C 180,E1 22622.804,E2 22622.804} C_VEL
LIN {X 0,Y 150.957,Z 883.128,A -85,B 0,C 180,E1 22637.854,E2 22637.854} C_VEL
LIN {X 0,Y 162.261,Z 853.212,A -85,B 0,C 180,E1 22644.263,E2 22644.263} C_VEL
LIN {X 0,Y 155.296,Z 815.225,A -85,B 0,C 180,E1 22655.084,E2 22655.084} C_VEL
LIN {X 0,Y 141.158,Z 783.178,A -85,B 0,C 180,E1 22668.772,E2 22668.772} C_VEL
LIN {X 0,Y 132.432,Z 769.19,A -85,B 0,C 180,E1 22681.239,E2 22681.239} C_VEL
LIN {X 0,Y 129.003,Z 768.053,A -85,B 0,C 180,E1 22699.785,E2 22699.785} C_VEL
LIN {X 0,Y 132.58,Z 773.864,A -85,B 0,C 180,E1 22711.013,E2 22711.013} C_VEL
LIN {X 0,Y 142.488,Z 788.993,A -85,B 0,C 180,E1 22724.819,E2 22724.819} C_VEL
LIN {X 0,Y 153.346,Z 816.741,A -85,B 0,C 180,E1 22737.887,E2 22737.887} C_VEL
LIN {X 0,Y 156.034,Z 846.419,A -85,B 0,C 180,E1 22748.455,E2 22748.455} C_VEL
LIN {X 0,Y 140.703,Z 880.122,A -85,B 0,C 180,E1 22760.687,E2 22760.687} C_VEL
LIN {X 0,Y 129.483,Z 902.032,A -85,B 0,C 180,E1 22778.279,E2 22778.279} C_VEL
LIN {X 0,Y 129.582,Z 910.71,A -85,B 0,C 180,E1 22798.54,E2 22798.54} C_VEL
LIN {X 0,Y 133.42,Z 910.457,A -85,B 0,C 180,E1 22806.497,E2 22806.497} C_VEL
LIN {X 0,Y 139.069,Z 906.494,A -85,B 0,C 180,E1 22821.157,E2 22821.157} C_VEL
LIN {X 0,Y 166.127,Z 886.093,A -85,B 0,C 180,E1 22835.506,E2 22835.506} C_VEL
LIN {X 0,Y 174.178,Z 877.269,A -85,B 0,C 180,E1 22839.033,E2 22839.033} C_VEL
LIN {X 0,Y 180.49,Z 862.196,A -85,B 0,C 180,E1 22849.55,E2 22849.55} C_VEL
LIN {X 0,Y 184.468,Z 851.828,A -85,B 0,C 180,E1 22862.351,E2 22862.351} C_VEL
LIN {X 0,Y 185.019,Z 857.963,A -85,B 0,C 180,E1 22874.239,E2 22874.239} C_VEL
LIN {X 0,Y 185.121,Z 874.532,A -85,B 0,C 180,E1 22885.73,E2 22885.73} C_VEL
LIN {X 0,Y 180.518,Z 883.112,A -85,B 0,C 180,E1 22888.032,E2 22888.032} C_VEL
LIN {X 0,Y 150.055,Z 917.046,A -85,B 0,C 180,E1 22898.394,E2 22898.394} C_VEL
LIN {X 0,Y 124.807,Z 938.559,A -85,B 0,C 180,E1 22916.829,E2 22916.829} C_VEL
LIN {X 0,Y 117.674,Z 945.943,A -85,B 0,C 180,E1 22938.848,E2 22938.848} C_VEL
LIN {X 0,Y 118.795,Z 944.138,A -85,B 0,C 180,E1 22953.665,E2 22953.665} C_VEL
LIN {X 0,Y 120.813,Z 928.433,A -85,B 0,C 180,E1 22976.084,E2 22976.084} C_VEL
LIN {X 0,Y 136.374,Z 898.187,A -85,B 0,C 180,E1 22994.444,E2 22994.444} C_VEL
LIN {X 0,Y 155.607,Z 856.34,A -85,B 0,C 180,E1 23005.394,E2 23005.394} C_VEL
LIN {X 0,Y 149.856,Z 818.939,A -85,B 0,C 180,E1 23016.903,E2 23016.903} C_VEL
LIN {X 0,Y 137.73,Z 788.711,A -85,B 0,C 180,E1 23030.999,E2 23030.999} C_VEL
LIN {X 0,Y 130.565,Z 776.415,A -85,B 0,C 180,E1 23043.027,E2 23043.027} C_VEL
LIN {X 0,Y 128.483,Z 776.844,A -85,B 0,C 180,E1 23062.7,E2 23062.7} C_VEL
LIN {X 0,Y 135.356,Z 788.838,A -85,B 0,C 180,E1 23078.329,E2 23078.329} C_VEL
LIN {X 0,Y 145.855,Z 813.451,A -85,B 0,C 180,E1 23093.119,E2 23093.119} C_VEL
LIN {X 0,Y 149.747,Z 842.366,A -85,B 0,C 180,E1 23104.628,E2 23104.628} C_VEL
LIN {X 0,Y 145.469,Z 858.538,A -85,B 0,C 180,E1 23109.953,E2 23109.953} C_VEL
LIN {X 0,Y 128.761,Z 889.602,A -85,B 0,C 180,E1 23124.614,E2 23124.614} C_VEL
LIN {X 0,Y 120.128,Z 907.292,A -85,B 0,C 180,E1 23144.547,E2 23144.547} C_VEL
LIN {X 0,Y 125.857,Z 911.805,A -85,B 0,C 180,E1 23167.476,E2 23167.476} C_VEL
LIN {X 0,Y 139.069,Z 906.494,A -85,B 0,C 180,E1 23181.157,E2 23181.157} C_VEL
LIN {X 0,Y 151.285,Z 896.024,A -85,B 0,C 180,E1 23193.656,E2 23193.656} C_VEL
LIN {X 0,Y 168.687,Z 880.157,A -85,B 0,C 180,E1 23200.838,E2 23200.838} C_VEL
LIN {X 0,Y 176.084,Z 865.257,A -85,B 0,C 180,E1 23212.566,E2 23212.566} C_VEL
LIN {X 0,Y 179.763,Z 858.42,A -85,B 0,C 180,E1 23222.413,E2 23222.413} C_VEL
LIN {X 0,Y 180.095,Z 864.577,A -85,B 0,C 180,E1 23234.298,E2 23234.298} C_VEL
LIN {X 0,Y 179.256,Z 879.125,A -85,B 0,C 180,E1 23244.823,E2 23244.823} C_VEL
LIN {X 0,Y 148.428,Z 913.476,A -85,B 0,C 180,E1 23254.489,E2 23254.489} C_VEL
LIN {X 0,Y 119.52,Z 936.471,A -85,B 0,C 180,E1 23272.909,E2 23272.909} C_VEL
LIN {X 0,Y 109.742,Z 944.698,A -85,B 0,C 180,E1 23298.031,E2 23298.031} C_VEL
LIN {X 0,Y 110.813,Z 942.757,A -85,B 0,C 180,E1 23313.929,E2 23313.929} C_VEL
LIN {X 0,Y 113.434,Z 926.618,A -85,B 0,C 180,E1 23337.923,E2 23337.923} C_VEL
LIN {X 0,Y 130.275,Z 896.221,A -85,B 0,C 180,E1 23356.767,E2 23356.767} C_VEL
LIN {X 0,Y 148.93,Z 856.843,A -85,B 0,C 180,E1 23367.375,E2 23367.375} C_VEL
LIN {X 0,Y 144.27,Z 821.596,A -85,B 0,C 180,E1 23379.214,E2 23379.214} C_VEL
LIN {X 0,Y 134.121,Z 794,A -85,B 0,C 180,E1 23393.53,E2 23393.53} C_VEL
LIN {X 0,Y 128.729,Z 783.71,A -85,B 0,C 180,E1 23404.742,E2 23404.742} C_VEL
LIN {X 0,Y 128.137,Z 785.914,A -85,B 0,C 180,E1 23426.253,E2 23426.253} C_VEL
LIN {X 0,Y 136.079,Z 804.159,A -85,B 0,C 180,E1 23443.537,E2 23443.537} C_VEL
LIN {X 0,Y 142.684,Z 828.68,A -85,B 0,C 180,E1 23456.327,E2 23456.327} C_VEL
LIN {X 0,Y 141.834,Z 854.145,A -85,B 0,C 180,E1 23466.487,E2 23466.487} C_VEL
LIN {X 0,Y 124.047,Z 886.357,A -85,B 0,C 180,E1 23480.308,E2 23480.308} C_VEL
LIN {X 0,Y 112.608,Z 906.902,A -85,B 0,C 180,E1 23501.66,E2 23501.66} C_VEL
LIN {X 0,Y 116.692,Z 913.353,A -85,B 0,C 180,E1 23525.816,E2 23525.816} C_VEL
LIN {X 0,Y 137.114,Z 905.511,A -85,B 0,C 180,E1 23546.105,E2 23546.105} C_VEL
LIN {X 0,Y 151.285,Z 896.024,A -85,B 0,C 180,E1 23553.656,E2 23553.656} C_VEL
LIN {X 0,Y 162.237,Z 884.554,A -85,B 0,C 180,E1 23561.565,E2 23561.565} C_VEL
LIN {X 0,Y 164.812,Z 880.829,A -85,B 0,C 180,E1 23564.332,E2 23564.332} C_VEL
LIN {X 0,Y 171.536,Z 869.357,A -85,B 0,C 180,E1 23574.918,E2 23574.918} C_VEL
LIN {X 0,Y 174.791,Z 864.85,A -85,B 0,C 180,E1 23583.211,E2 23583.211} C_VEL
LIN {X 0,Y 174.755,Z 872.875,A -85,B 0,C 180,E1 23596.21,E2 23596.21} C_VEL
LIN {X 0,Y 172.563,Z 883.729,A -85,B 0,C 180,E1 23603.531,E2 23603.531} C_VEL
LIN {X 0,Y 139.594,Z 916.5,A -85,B 0,C 180,E1 23613.545,E2 23613.545} C_VEL
LIN {X 0,Y 111.422,Z 936.616,A -85,B 0,C 180,E1 23632.203,E2 23632.203} C_VEL
LIN {X 0,Y 101.811,Z 943.449,A -85,B 0,C 180,E1 23657.083,E2 23657.083} C_VEL
LIN {X 0,Y 102.814,Z 941.343,A -85,B 0,C 180,E1 23674.235,E2 23674.235} C_VEL
LIN {X 0,Y 106.235,Z 924.742,A -85,B 0,C 180,E1 23700.001,E2 23700.001} C_VEL
LIN {X 0,Y 124.992,Z 893.281,A -85,B 0,C 180,E1 23719.669,E2 23719.669} C_VEL
LIN {X 0,Y 142.387,Z 857.245,A -85,B 0,C 180,E1 23729.595,E2 23729.595} C_VEL
LIN {X 0,Y 138.295,Z 822.659,A -85,B 0,C 180,E1 23742.445,E2 23742.445} C_VEL
LIN {X 0,Y 129.935,Z 797.126,A -85,B 0,C 180,E1 23757.76,E2 23757.76} C_VEL
LIN {X 0,Y 125.919,Z 790.477,A -85,B 0,C 180,E1 23769.547,E2 23769.547} C_VEL
LIN {X 0,Y 126.639,Z 796.26,A -85,B 0,C 180,E1 23788.282,E2 23788.282} C_VEL
LIN {X 0,Y 133.006,Z 812.758,A -85,B 0,C 180,E1 23803.887,E2 23803.887} C_VEL
LIN {X 0,Y 137.381,Z 839.037,A -85,B 0,C 180,E1 23817.576,E2 23817.576} C_VEL
LIN {X 0,Y 134.344,Z 857.666,A -85,B 0,C 180,E1 23825.09,E2 23825.09} C_VEL
LIN {X 0,Y 115.573,Z 889.395,A -85,B 0,C 180,E1 23840.052,E2 23840.052} C_VEL
LIN {X 0,Y 104.485,Z 908.606,A -85,B 0,C 180,E1 23862.581,E2 23862.581} C_VEL
LIN {X 0,Y 109.972,Z 914.527,A -85,B 0,C 180,E1 23888.385,E2 23888.385} C_VEL
LIN {X 0,Y 132.57,Z 906.224,A -85,B 0,C 180,E1 23909.15,E2 23909.15} C_VEL
LIN {X 0,Y 162.824,Z 883.632,A -85,B 0,C 180,E1 23922.27,E2 23922.27} C_VEL
LIN {X 0,Y 164.812,Z 880.829,A -85,B 0,C 180,E1 23924.332,E2 23924.332} C_VEL
LIN {X 0,Y 165.718,Z 875.806,A -85,B 0,C 180,E1 23933.432,E2 23933.432} C_VEL
LIN {X 0,Y 166.466,Z 874.253,A -85,B 0,C 180,E1 23936.545,E2 23936.545} C_VEL
LIN {X 0,Y 169.465,Z 870.932,A -85,B 0,C 180,E1 23942.56,E2 23942.56} C_VEL
LIN {X 0,Y 169.255,Z 877.394,A -85,B 0,C 180,E1 23954.722,E2 23954.722} C_VEL
LIN {X 0,Y 166.635,Z 886.789,A -85,B 0,C 180,E1 23961.631,E2 23961.631} C_VEL
LIN {X 0,Y 131.971,Z 918.294,A -85,B 0,C 180,E1 23972.001,E2 23972.001} C_VEL
LIN {X 0,Y 101.815,Z 937.491,A -85,B 0,C 180,E1 23993.41,E2 23993.41} C_VEL
LIN {X 0,Y 94.546,Z 941.903,A -85,B 0,C 180,E1 24025.4,E2 24025.4} C_VEL
LIN {X 0,Y 94.433,Z 935.933,A -85,B 0,C 180,E1 24043.952,E2 24043.952} C_VEL
LIN {X 0,Y 105.189,Z 913.51,A -85,B 0,C 180,E1 24070.486,E2 24070.486} C_VEL
LIN {X 0,Y 127.646,Z 877.402,A -85,B 0,C 180,E1 24086.96,E2 24086.96} C_VEL
LIN {X 0,Y 135.923,Z 859.022,A -85,B 0,C 180,E1 24091.574,E2 24091.574} C_VEL
LIN {X 0,Y 133.461,Z 827.398,A -85,B 0,C 180,E1 24104.249,E2 24104.249} C_VEL
LIN {X 0,Y 126.946,Z 803.4,A -85,B 0,C 180,E1 24119.79,E2 24119.79} C_VEL
LIN {X 0,Y 123.555,Z 798.346,A -85,B 0,C 180,E1 24132.731,E2 24132.731} C_VEL
LIN {X 0,Y 124.1,Z 803.515,A -85,B 0,C 180,E1 24147.304,E2 24147.304} C_VEL
LIN {X 0,Y 128.877,Z 819.204,A -85,B 0,C 180,E1 24162.831,E2 24162.831} C_VEL
LIN {X 0,Y 131.372,Z 844.372,A -85,B 0,C 180,E1 24176.715,E2 24176.715} C_VEL
LIN {X 0,Y 127.739,Z 859.813,A -85,B 0,C 180,E1 24183.156,E2 24183.156} C_VEL
LIN {X 0,Y 107.552,Z 891.677,A -85,B 0,C 180,E1 24199.302,E2 24199.302} C_VEL
LIN {X 0,Y 96.369,Z 910.298,A -85,B 0,C 180,E1 24223.66,E2 24223.66} C_VEL
LIN {X 0,Y 103.475,Z 915.68,A -85,B 0,C 180,E1 24251.294,E2 24251.294} C_VEL
LIN {X 0,Y 128.43,Z 906.929,A -85,B 0,C 180,E1 24272.398,E2 24272.398} C_VEL
LIN {X 0,Y 158.142,Z 885.774,A -85,B 0,C 180,E1 24284.839,E2 24284.839} C_VEL
LIN {X 0,Y 166.466,Z 874.253,A -85,B 0,C 180,E1 24296.545,E2 24296.545} C_VEL
LIN {X 0,Y 163.789,Z 877.417,A -85,B 0,C 180,E1 24304.753,E2 24304.753} C_VEL
LIN {X 0,Y 162.833,Z 885.726,A -85,B 0,C 180,E1 24317.183,E2 24317.183} C_VEL
LIN {X 0,Y 159.407,Z 891.168,A -85,B 0,C 180,E1 24319.892,E2 24319.892} C_VEL
LIN {X 0,Y 123.498,Z 920.519,A -85,B 0,C 180,E1 24330.668,E2 24330.668} C_VEL
LIN {X 0,Y 95.344,Z 936.436,A -85,B 0,C 180,E1 24350.459,E2 24350.459} C_VEL
LIN {X 0,Y 86.555,Z 940.563,A -85,B 0,C 180,E1 24384.974,E2 24384.974} C_VEL
LIN {X 0,Y 86.588,Z 934.217,A -85,B 0,C 180,E1 24405.482,E2 24405.482} C_VEL
LIN {X 0,Y 99.916,Z 910.285,A -85,B 0,C 180,E1 24434.404,E2 24434.404} C_VEL
LIN {X 0,Y 124.107,Z 873.053,A -85,B 0,C 180,E1 24450.495,E2 24450.495} C_VEL
LIN {X 0,Y 129.79,Z 858.236,A -85,B 0,C 180,E1 24454.682,E2 24454.682} C_VEL
LIN {X 0,Y 127.988,Z 828.55,A -85,B 0,C 180,E1 24468.033,E2 24468.033} C_VEL
LIN {X 0,Y 123.463,Z 807.544,A -85,B 0,C 180,E1 24483.974,E2 24483.974} C_VEL
LIN {X 0,Y 120.922,Z 807.32,A -85,B 0,C 180,E1 24499.73,E2 24499.73} C_VEL
LIN {X 0,Y 123.72,Z 820.595,A -85,B 0,C 180,E1 24517.909,E2 24517.909} C_VEL
LIN {X 0,Y 125.706,Z 842.517,A -85,B 0,C 180,E1 24532.09,E2 24532.09} C_VEL
LIN {X 0,Y 121.864,Z 860.942,A -85,B 0,C 180,E1 24540.722,E2 24540.722} C_VEL
LIN {X 0,Y 100.813,Z 892.226,A -85,B 0,C 180,E1 24556.947,E2 24556.947} C_VEL
LIN {X 0,Y 88.306,Z 911.939,A -85,B 0,C 180,E1 24584.935,E2 24584.935} C_VEL
LIN {X 0,Y 98.432,Z 916.728,A -85,B 0,C 180,E1 24616.055,E2 24616.055} C_VEL
LIN {X 0,Y 127.305,Z 906.257,A -85,B 0,C 180,E1 24637.083,E2 24637.083} C_VEL
LIN {X 0,Y 153.227,Z 888.461,A -85,B 0,C 180,E1 24647.197,E2 24647.197} C_VEL
LIN {X 0,Y 162.003,Z 878.458,A -85,B 0,C 180,E1 24659.223,E2 24659.223} C_VEL
LIN {X 0,Y 163.789,Z 877.417,A -85,B 0,C 180,E1 24664.753,E2 24664.753} C_VEL
LIN {X 0,Y 157.288,Z 888.808,A -85,B 0,C 180,E1 24674.924,E2 24674.924} C_VEL
LIN {X 0,Y 156.673,Z 890.462,A -85,B 0,C 180,E1 24676.469,E2 24676.469} C_VEL
LIN {X 0,Y 119.538,Z 919.788,A -85,B 0,C 180,E1 24687.298,E2 24687.298} C_VEL
LIN {X 0,Y 89.165,Z 935.389,A -85,B 0,C 180,E1 24707.099,E2 24707.099} C_VEL
LIN {X 0,Y 78.545,Z 939.218,A -85,B 0,C 180,E1 24744.46,E2 24744.46} C_VEL
LIN {X 0,Y 78.753,Z 932.727,A -85,B 0,C 180,E1 24766.805,E2 24766.805} C_VEL
LIN {X 0,Y 93.286,Z 909.273,A -85,B 0,C 180,E1 24797.064,E2 24797.064} C_VEL
LIN {X 0,Y 118.759,Z 872.373,A -85,B 0,C 180,E1 24813.291,E2 24813.291} C_VEL
LIN {X 0,Y 123.66,Z 860.106,A -85,B 0,C 180,E1 24816.992,E2 24816.992} C_VEL
LIN {X 0,Y 123.133,Z 831.487,A -85,B 0,C 180,E1 24831.147,E2 24831.147} C_VEL
LIN {X 0,Y 120.379,Z 814.473,A -85,B 0,C 180,E1 24845.76,E2 24845.76} C_VEL
LIN {X 0,Y 118.265,Z 817.31,A -85,B 0,C 180,E1 24864.658,E2 24864.658} C_VEL
LIN {X 0,Y 120.178,Z 832.297,A -85,B 0,C 180,E1 24881.029,E2 24881.029} C_VEL
LIN {X 0,Y 118.913,Z 855.052,A -85,B 0,C 180,E1 24894.947,E2 24894.947} C_VEL
LIN {X 0,Y 109.007,Z 872.845,A -85,B 0,C 180,E1 24901.972,E2 24901.972} C_VEL
LIN {X 0,Y 87.799,Z 900.824,A -85,B 0,C 180,E1 24922.548,E2 24922.548} C_VEL
LIN {X 0,Y 80.325,Z 914.859,A -85,B 0,C 180,E1 24950.727,E2 24950.727} C_VEL
LIN {X 0,Y 91.464,Z 917.985,A -85,B 0,C 180,E1 24978.296,E2 24978.296} C_VEL
LIN {X 0,Y 121.508,Z 908.276,A -85,B 0,C 180,E1 24999.5,E2 24999.5} C_VEL
LIN {X 0,Y 148.277,Z 891.28,A -85,B 0,C 180,E1 25009.605,E2 25009.605} C_VEL
LIN {X 0,Y 156.051,Z 883.94,A -85,B 0,C 180,E1 25019.631,E2 25019.631} C_VEL
LIN {X 0,Y 157.879,Z 883.06,A -85,B 0,C 180,E1 25024.567,E2 25024.567} C_VEL
LIN {X 0,Y 156.673,Z 890.462,A -85,B 0,C 180,E1 25036.469,E2 25036.469} C_VEL
LIN {X 0,Y 149.161,Z 897.16,A -85,B 0,C 180,E1 25037.618,E2 25037.618} C_VEL
LIN {X 0,Y 137.656,Z 904.821,A -85,B 0,C 180,E1 25037.578,E2 25037.578} C_VEL
LIN {X 0,Y 98.159,Z 928.242,A -85,B 0,C 180,E1 25051.759,E2 25051.759} C_VEL
LIN {X 0,Y 73.533,Z 937.7,A -85,B 0,C 180,E1 25078.943,E2 25078.943} C_VEL
LIN {X 0,Y 70.859,Z 936.96,A -85,B 0,C 180,E1 25110.004,E2 25110.004} C_VEL
LIN {X 0,Y 74.454,Z 923.696,A -85,B 0,C 180,E1 25143.02,E2 25143.02} C_VEL
LIN {X 0,Y 97.827,Z 894.385,A -85,B 0,C 180,E1 25168.568,E2 25168.568} C_VEL
LIN {X 0,Y 117.451,Z 864.146,A -85,B 0,C 180,E1 25178.512,E2 25178.512} C_VEL
LIN {X 0,Y 118.635,Z 837.287,A -85,B 0,C 180,E1 25192.66,E2 25192.66} C_VEL
LIN {X 0,Y 117.376,Z 822.136,A -85,B 0,C 180,E1 25205.908,E2 25205.908} C_VEL
LIN {X 0,Y 115.201,Z 823.264,A -85,B 0,C 180,E1 25222.134,E2 25222.134} C_VEL
LIN {X 0,Y 115.527,Z 837.679,A -85,B 0,C 180,E1 25239.245,E2 25239.245} C_VEL
LIN {X 0,Y 112.996,Z 858.282,A -85,B 0,C 180,E1 25252.814,E2 25252.814} C_VEL
LIN {X 0,Y 90.132,Z 890.719,A -85,B 0,C 180,E1 25269.052,E2 25269.052} C_VEL
LIN {X 0,Y 73.163,Z 912.025,A -85,B 0,C 180,E1 25298.946,E2 25298.946} C_VEL
LIN {X 0,Y 78.734,Z 919.312,A -85,B 0,C 180,E1 25332.419,E2 25332.419} C_VEL
LIN {X 0,Y 106.612,Z 914.02,A -85,B 0,C 180,E1 25357.699,E2 25357.699} C_VEL
LIN {X 0,Y 141.963,Z 895.413,A -85,B 0,C 180,E1 25370.765,E2 25370.765} C_VEL
LIN {X 0,Y 151.77,Z 888.019,A -85,B 0,C 180,E1 25382.858,E2 25382.858} C_VEL
LIN {X 0,Y 151.159,Z 892.602,A -85,B 0,C 180,E1 25393.048,E2 25393.048} C_VEL
LIN {X 0,Y 147.644,Z 896.801,A -85,B 0,C 180,E1 25395.51,E2 25395.51} C_VEL
LIN {X 0,Y 137.656,Z 904.821,A -85,B 0,C 180,E1 25397.578,E2 25397.578} C_VEL
LIN {X 0,Y 107.505,Z 921.234,A -85,B 0,C 180,E1 25401.772,E2 25401.772} C_VEL
LIN {X 0,Y 73.525,Z 934.66,A -85,B 0,C 180,E1 25423.752,E2 25423.752} C_VEL
LIN {X 0,Y 62.538,Z 936.5,A -85,B 0,C 180,E1 25463.035,E2 25463.035} C_VEL
LIN {X 0,Y 62.758,Z 931.452,A -85,B 0,C 180,E1 25485.564,E2 25485.564} C_VEL
LIN {X 0,Y 79.239,Z 908.865,A -85,B 0,C 180,E1 25522.193,E2 25522.193} C_VEL
LIN {X 0,Y 107.008,Z 874.078,A -85,B 0,C 180,E1 25538.904,E2 25538.904} C_VEL
LIN {X 0,Y 112.374,Z 861.695,A -85,B 0,C 180,E1 25543.43,E2 25543.43} C_VEL
LIN {X 0,Y 114.061,Z 838.168,A -85,B 0,C 180,E1 25557.852,E2 25557.852} C_VEL
LIN {X 0,Y 113.653,Z 828.775,A -85,B 0,C 180,E1 25568.285,E2 25568.285} C_VEL
LIN {X 0,Y 111.363,Z 832.66,A -85,B 0,C 180,E1 25585.043,E2 25585.043} C_VEL
LIN {X 0,Y 110.351,Z 847.194,A -85,B 0,C 180,E1 25600.85,E2 25600.85} C_VEL
LIN {X 0,Y 105.172,Z 865.275,A -85,B 0,C 180,E1 25612.172,E2 25612.172} C_VEL
LIN {X 0,Y 79.235,Z 896.572,A -85,B 0,C 180,E1 25630.262,E2 25630.262} C_VEL
LIN {X 0,Y 64.578,Z 914.807,A -85,B 0,C 180,E1 25663.576,E2 25663.576} C_VEL
LIN {X 0,Y 72.74,Z 920.566,A -85,B 0,C 180,E1 25696.898,E2 25696.898} C_VEL
LIN {X 0,Y 103.693,Z 914.832,A -85,B 0,C 180,E1 25722.035,E2 25722.035} C_VEL
LIN {X 0,Y 137.224,Z 898.255,A -85,B 0,C 180,E1 25733.386,E2 25733.386} C_VEL
LIN {X 0,Y 145.332,Z 893.18,A -85,B 0,C 180,E1 25742.985,E2 25742.985} C_VEL
LIN {X 0,Y 144.863,Z 896.773,A -85,B 0,C 180,E1 25751.938,E2 25751.938} C_VEL
LIN {X 0,Y 107.505,Z 921.234,A -85,B 0,C 180,E1 25761.772,E2 25761.772} C_VEL
LIN {X 0,Y 76.711,Z 931.188,A -85,B 0,C 180,E1 25770.938,E2 25770.938} C_VEL
LIN {X 0,Y 54.322,Z 935.384,A -85,B 0,C 180,E1 25817.8,E2 25817.8} C_VEL
LIN {X 0,Y 54.864,Z 932.526,A -85,B 0,C 180,E1 25837.955,E2 25837.955} C_VEL
LIN {X 0,Y 68.175,Z 912.925,A -85,B 0,C 180,E1 25881.185,E2 25881.185} C_VEL
LIN {X 0,Y 98.316,Z 879.238,A -85,B 0,C 180,E1 25900.995,E2 25900.995} C_VEL
LIN {X 0,Y 106.492,Z 865.444,A -85,B 0,C 180,E1 25905.502,E2 25905.502} C_VEL
LIN {X 0,Y 109.788,Z 842.384,A -85,B 0,C 180,E1 25920.895,E2 25920.895} C_VEL
LIN {X 0,Y 110.132,Z 836.169,A -85,B 0,C 180,E1 25927.93,E2 25927.93} C_VEL
LIN {X 0,Y 107.549,Z 839.063,A -85,B 0,C 180,E1 25943.476,E2 25943.476} C_VEL
LIN {X 0,Y 105.469,Z 851.519,A -85,B 0,C 180,E1 25958.352,E2 25958.352} C_VEL
LIN {X 0,Y 99.655,Z 867.395,A -85,B 0,C 180,E1 25968.946,E2 25968.946} C_VEL
LIN {X 0,Y 71.083,Z 899.285,A -85,B 0,C 180,E1 25988.575,E2 25988.575} C_VEL
LIN {X 0,Y 56.467,Z 917.441,A -85,B 0,C 180,E1 26029.786,E2 26029.786} C_VEL
LIN {X 0,Y 76.991,Z 921.3,A -85,B 0,C 180,E1 26072.49,E2 26072.49} C_VEL
LIN {X 0,Y 115.116,Z 910.328,A -85,B 0,C 180,E1 26091.372,E2 26091.372} C_VEL
LIN {X 0,Y 133.157,Z 900.851,A -85,B 0,C 180,E1 26096.725,E2 26096.725} C_VEL
LIN {X 0,Y 138.665,Z 898.033,A -85,B 0,C 180,E1 26103.129,E2 26103.129} C_VEL
LIN {X 0,Y 137.379,Z 901.212,A -85,B 0,C 180,E1 26110.31,E2 26110.31} C_VEL
LIN {X 0,Y 93.818,Z 925.22,A -85,B 0,C 180,E1 26121.558,E2 26121.558} C_VEL
LIN {X 0,Y 76.711,Z 931.188,A -85,B 0,C 180,E1 26130.938,E2 26130.938} C_VEL
LIN {X 0,Y 50.59,Z 934.287,A -85,B 0,C 180,E1 26152.86,E2 26152.86} C_VEL
LIN {X 0,Y 47.113,Z 932.678,A -85,B 0,C 180,E1 26190.006,E2 26190.006} C_VEL
LIN {X 0,Y 58.149,Z 915.535,A -85,B 0,C 180,E1 26241.059,E2 26241.059} C_VEL
LIN {X 0,Y 89,Z 884.826,A -85,B 0,C 180,E1 26263.093,E2 26263.093} C_VEL
LIN {X 0,Y 100.818,Z 868.568,A -85,B 0,C 180,E1 26268.09,E2 26268.09} C_VEL
LIN {X 0,Y 105.437,Z 847.685,A -85,B 0,C 180,E1 26283.104,E2 26283.104} C_VEL
LIN {X 0,Y 106.132,Z 843.26,A -85,B 0,C 180,E1 26288.231,E2 26288.231} C_VEL
LIN {X 0,Y 103.157,Z 846.741,A -85,B 0,C 180,E1 26304.54,E2 26304.54} C_VEL
LIN {X 0,Y 98.825,Z 861.161,A -85,B 0,C 180,E1 26320.186,E2 26320.186} C_VEL
LIN {X 0,Y 93.611,Z 870.509,A -85,B 0,C 180,E1 26325.639,E2 26325.639} C_VEL
LIN {X 0,Y 63.891,Z 901.093,A -85,B 0,C 180,E1 26345.434,E2 26345.434} C_VEL
LIN {X 0,Y 48.61,Z 918.784,A -85,B 0,C 180,E1 26391.854,E2 26391.854} C_VEL
LIN {X 0,Y 62.465,Z 923.017,A -85,B 0,C 180,E1 26428.238,E2 26428.238} C_VEL
LIN {X 0,Y 99.782,Z 916.506,A -85,B 0,C 180,E1 26451.313,E2 26451.313} C_VEL
LIN {X 0,Y 125.708,Z 905.349,A -85,B 0,C 180,E1 26458.168,E2 26458.168} C_VEL
LIN {X 0,Y 131.699,Z 902.625,A -85,B 0,C 180,E1 26463.295,E2 26463.295} C_VEL
LIN {X 0,Y 128.357,Z 905.922,A -85,B 0,C 180,E1 26468.051,E2 26468.051} C_VEL
LIN {X 0,Y 82.845,Z 927.254,A -85,B 0,C 180,E1 26480.039,E2 26480.039} C_VEL
LIN {X 0,Y 50.59,Z 934.287,A -85,B 0,C 180,E1 26512.86,E2 26512.86} C_VEL
LIN {X 0,Y 40.073,Z 932.069,A -85,B 0,C 180,E1 26544.42,E2 26544.42} C_VEL
LIN {X 0,Y 38.829,Z 930.054,A -85,B 0,C 180,E1 26557.262,E2 26557.262} C_VEL
LIN {X 0,Y 57.816,Z 909.937,A -85,B 0,C 180,E1 26612.371,E2 26612.371} C_VEL
LIN {X 0,Y 91.142,Z 877.005,A -85,B 0,C 180,E1 26629.628,E2 26629.628} C_VEL
LIN {X 0,Y 96.684,Z 867.691,A -85,B 0,C 180,E1 26633.536,E2 26633.536} C_VEL
LIN {X 0,Y 101.325,Z 851.784,A -85,B 0,C 180,E1 26646.676,E2 26646.676} C_VEL
LIN {X 0,Y 100.042,Z 850.66,A -85,B 0,C 180,E1 26657.677,E2 26657.677} C_VEL
LIN {X 0,Y 96.269,Z 859.286,A -85,B 0,C 180,E1 26671.858,E2 26671.858} C_VEL
LIN {X 0,Y 89.656,Z 871.589,A -85,B 0,C 180,E1 26681.308,E2 26681.308} C_VEL
LIN {X 0,Y 57.891,Z 902.155,A -85,B 0,C 180,E1 26700.554,E2 26700.554} C_VEL
LIN {X 0,Y 40.638,Z 919.48,A -85,B 0,C 180,E1 26750.924,E2 26750.924} C_VEL
LIN {X 0,Y 61.963,Z 924.164,A -85,B 0,C 180,E1 26798.428,E2 26798.428} C_VEL
LIN {X 0,Y 102.557,Z 916.037,A -85,B 0,C 180,E1 26817.169,E2 26817.169} C_VEL
LIN {X 0,Y 120.533,Z 908.512,A -85,B 0,C 180,E1 26821.089,E2 26821.089} C_VEL
LIN {X 0,Y 124.838,Z 906.865,A -85,B 0,C 180,E1 26824.19,E2 26824.19} C_VEL
LIN {X 0,Y 78.638,Z 926.814,A -85,B 0,C 180,E1 26835.236,E2 26835.236} C_VEL
LIN {X 0,Y 41.088,Z 933.184,A -85,B 0,C 180,E1 26876.365,E2 26876.365} C_VEL
LIN {X 0,Y 38.829,Z 930.054,A -85,B 0,C 180,E1 26917.262,E2 26917.262} C_VEL
LIN {X 0,Y 41.313,Z 917.368,A -85,B 0,C 180,E1 26966.183,E2 26966.183} C_VEL
LIN {X 0,Y 76.807,Z 888.502,A -85,B 0,C 180,E1 26991.108,E2 26991.108} C_VEL
LIN {X 0,Y 91.463,Z 871.167,A -85,B 0,C 180,E1 26996.563,E2 26996.563} C_VEL
LIN {X 0,Y 96.971,Z 856.603,A -85,B 0,C 180,E1 27010.266,E2 27010.266} C_VEL
LIN {X 0,Y 92.816,Z 861.56,A -85,B 0,C 180,E1 27025.931,E2 27025.931} C_VEL
LIN {X 0,Y 87.124,Z 871.662,A -85,B 0,C 180,E1 27036.4,E2 27036.4} C_VEL
LIN {X 0,Y 52.379,Z 903.184,A -85,B 0,C 180,E1 27054.581,E2 27054.581} C_VEL
LIN {X 0,Y 32.976,Z 921.058,A -85,B 0,C 180,E1 27116.111,E2 27116.111} C_VEL
LIN {X 0,Y 55.486,Z 925.473,A -85,B 0,C 180,E1 27163.172,E2 27163.172} C_VEL
LIN {X 0,Y 98.654,Z 918.088,A -85,B 0,C 180,E1 27181.052,E2 27181.052} C_VEL
LIN {X 0,Y 105.714,Z 915.654,A -85,B 0,C 180,E1 27182.508,E2 27182.508} C_VEL
LIN {X 0,Y 56.088,Z 930.216,A -85,B 0,C 180,E1 27198.752,E2 27198.752} C_VEL
LIN {X 0,Y 30.782,Z 930.817,A -85,B 0,C 180,E1 27255.739,E2 27255.739} C_VEL
LIN {X 0,Y 31.258,Z 926.696,A -85,B 0,C 180,E1 27291.363,E2 27291.363} C_VEL
LIN {X 0,Y 41.313,Z 917.368,A -85,B 0,C 180,E1 27326.183,E2 27326.183} C_VEL
LIN {X 0,Y 61.152,Z 898.921,A -85,B 0,C 180,E1 27352.682,E2 27352.682} C_VEL
LIN {X 0,Y 86.772,Z 873.706,A -85,B 0,C 180,E1 27360.498,E2 27360.498} C_VEL
LIN {X 0,Y 91.641,Z 863.911,A -85,B 0,C 180,E1 27369.544,E2 27369.544} C_VEL
LIN {X 0,Y 88.328,Z 866.62,A -85,B 0,C 180,E1 27383.143,E2 27383.143} C_VEL
LIN {X 0,Y 82.323,Z 874.905,A -85,B 0,C 180,E1 27391.853,E2 27391.853} C_VEL
LIN {X 0,Y 45.963,Z 905.252,A -85,B 0,C 180,E1 27408.665,E2 27408.665} C_VEL
LIN {X 0,Y 26.144,Z 922.94,A -85,B 0,C 180,E1 27487.206,E2 27487.206} C_VEL
LIN {X 0,Y 53.737,Z 926.648,A -85,B 0,C 180,E1 27531.862,E2 27531.862} C_VEL
LIN {X 0,Y 81.014,Z 923.613,A -85,B 0,C 180,E1 27542.18,E2 27542.18} C_VEL
LIN {X 0,Y 40.372,Z 930.382,A -85,B 0,C 180,E1 27560.01,E2 27560.01} C_VEL
LIN {X 0,Y 22.939,Z 927.511,A -85,B 0,C 180,E1 27637.485,E2 27637.485} C_VEL
LIN {X 0,Y 50.518,Z 906.918,A -85,B 0,C 180,E1 27707.53,E2 27707.53} C_VEL
LIN {X 0,Y 61.152,Z 898.921,A -85,B 0,C 180,E1 27712.682,E2 27712.682} C_VEL
LIN {X 0,Y 75.051,Z 883.945,A -85,B 0,C 180,E1 27723.342,E2 27723.342} C_VEL
LIN {X 0,Y 83.617,Z 874.352,A -85,B 0,C 180,E1 27726.482,E2 27726.482} C_VEL
LIN {X 0,Y 85.983,Z 869.656,A -85,B 0,C 180,E1 27733.883,E2 27733.883} C_VEL
LIN {X 0,Y 79.951,Z 876.183,A -85,B 0,C 180,E1 27746.493,E2 27746.493} C_VEL
LIN {X 0,Y 41.936,Z 906.278,A -85,B 0,C 180,E1 27759.725,E2 27759.725} C_VEL
LIN {X 0,Y 16.974,Z 922.504,A -85,B 0,C 180,E1 27836.536,E2 27836.536} C_VEL
LIN {X 0,Y 53.136,Z 927.94,A -85,B 0,C 180,E1 27901.77,E2 27901.77} C_VEL
LIN {X 0,Y 14.96,Z 927.086,A -85,B 0,C 180,E1 27982.133,E2 27982.133} C_VEL
LIN {X 0,Y 41.988,Z 909.444,A -85,B 0,C 180,E1 28073.746,E2 28073.746} C_VEL
LIN {X 0,Y 75.051,Z 883.945,A -85,B 0,C 180,E1 28083.342,E2 28083.342} C_VEL
LIN {X 0,Y 79.072,Z 877.78,A -85,B 0,C 180,E1 28090.949,E2 28090.949} C_VEL
LIN {X 0,Y 77.906,Z 877.892,A -85,B 0,C 180,E1 28099.133,E2 28099.133} C_VEL
LIN {X 0,Y 58.238,Z 894.878,A -85,B 0,C 180,E1 28104.201,E2 28104.201} C_VEL
LIN {X 0,Y 17.95,Z 917.655,A -85,B 0,C 180,E1 28126.839,E2 28126.839} C_VEL
LIN {X 0,Y 27.576,Z 927.881,A -85,B 0,C 180,E1 28259.891,E2 28259.891} C_VEL
LIN {X 0,Y 7.466,Z 924.14,A -85,B 0,C 180,E1 28380.584,E2 28380.584} C_VEL
LIN {X 0,Y 49.648,Z 902.453,A -85,B 0,C 180,E1 28446.525,E2 28446.525} C_VEL
LIN {X 0,Y 79.242,Z 877.626,A -85,B 0,C 180,E1 28450.688,E2 28450.688} C_VEL
LIN {X 0,Y 77.906,Z 877.892,A -85,B 0,C 180,E1 28459.133,E2 28459.133} C_VEL
LIN {X 0,Y 68.444,Z 886.695,A -85,B 0,C 180,E1 28462.796,E2 28462.796} C_VEL
LIN {X 0,Y 45.394,Z 903.885,A -85,B 0,C 180,E1 28456.931,E2 28456.931} C_VEL
LIN {X 0,Y 8.056,Z 921.274,A -85,B 0,C 180,E1 28459.533,E2 28459.533} C_VEL
LIN {X 0,Y 52.891,Z 899.095,A -85,B 0,C 180,E1 28455.752,E2 28455.752} C_VEL
LIN {X 0,Y 55.378,Z 897.252,A -85,B 0,C 180,E1 28456.42,E2 28456.42} C_VEL
LIN {X 0,Y 45.394,Z 903.885,A -85,B 0,C 180,E1 28456.931,E2 28456.931} C_VEL
LIN {X 0,Y 44.42,Z 905.602,A -85,B 0,C 180,E1 28456.984,E2 28456.984} C_VEL
LIN {X 0,Y 44.42,Z 1007,A -85,B 0,C 180,E1 28456.984,E2 28456.984} C_VEL
LIN {X 0,Y 44.42,Z 1007,A -85,B 0,C 180,E1 28456.984,E2 28456.984}

